RoboDK station: Trabajo_AndreaCasal.rdk

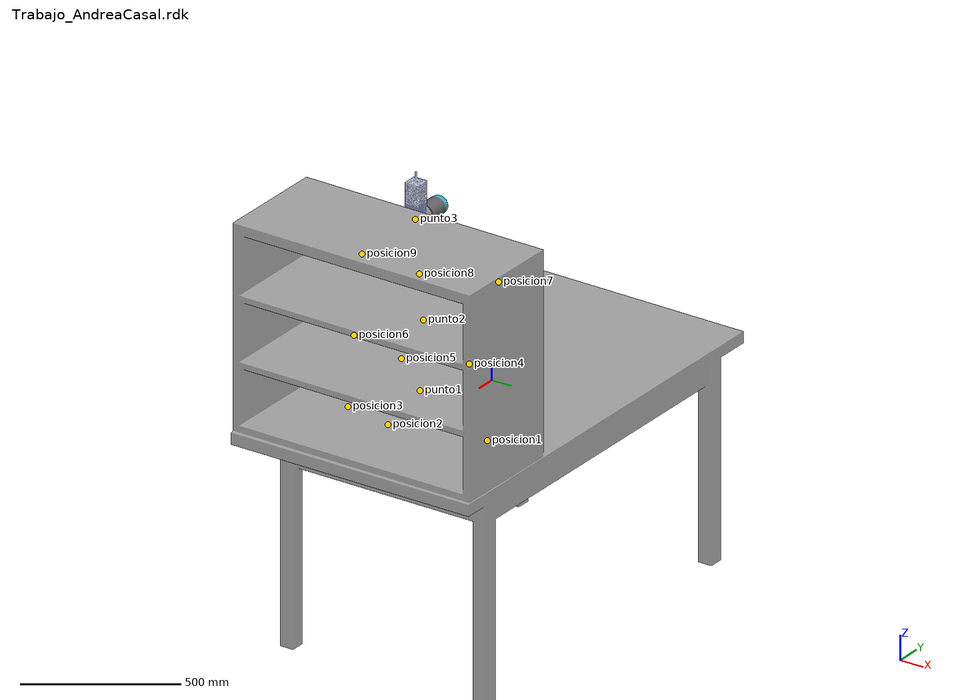
[picture v0: the station drawn from its stored meshes, robots at their saved joint values, targets as dots, program paths as lines]
Station Trabajo_AndreaCasal (saved by RoboDK 5.4.1). Poses are relative to the parent item; angles as X-Y-Z fixed-axis rotations.
  - frame UR3e Base at (447.56, 766.92, -5.55) mm, rotated rx 0 ry 0 rz -89.36 deg
    - robot UR3e: 6 axes, payload 3 kg, reach 500 mm, repeatability 0.03 mm, weight 11 kg
        modified DH rows (alpha deg, a mm, theta deg, d mm): 0, 0, 0, 151.9; 90, 0, 180, 0; 0, 243.55, 0, 0; 0, 213.2, 0, 131.05; -90, 0, 0, 85.35; 90, 0, 180, 92.1
        joint limits [-360, -360, -360, -360, -360, -360] to [360, 360, 360, 360, 360, 360]; home [0, -90, -90, 0, 90, 0]; saved at [-9.797, -78.984, -66.655, -34.361, 99.797, 0]
      - tool RGI-35-14-O-B, TCP at (0, 0, 3.37) mm, rotated rx 179.18 ry -0.35 rz -171.57 deg, size 50 x 211.5 x 50 mm, geometry from RGI-35-14-O-B.step
    - target punto1 (Cartesian target) at (291.92, -70.9, 62.1) mm, rotated rx 0 ry 0 rz -6.66 deg; joints [-219.826, -59.606, 132.901, -163.143, 270.876, 48.404] of UR3e
    - target punto2 (Cartesian target) at (275.14, -68.94, 300.54) mm, rotated rx 0 ry 0 rz -6.66 deg; joints [-221.915, -101.216, 99.747, -88.347, 270.87, 46.315] of UR3e
    - target punto3 (Cartesian target) at (200.73, -151.17, 596.64) mm, rotated rx -90.76 ry -8.43 rz 89.64 deg; joints [-9.797, -78.984, -66.655, -34.361, 99.797, 0] of UR3e
    - target posicion1 (Cartesian target) at (461.35, 299.35, 59.69) mm, rotated rx 0 ry 0 rz -96.24 deg; joints [46.918, -169.172, -22.416, -78.205, 89.136, 224.729] of UR3e
    - target posicion2 (Cartesian target) at (546.96, -17.63, 62.08) mm, rotated rx -0.01 ry 0.01 rz -96.16 deg; joints [12.113, 168.263, -333.534, 255.925, 89.422, 189.837] of UR3e
    - target posicion3 (Cartesian target) at (477.2, -215.05, 41.8) mm, rotated rx -1.06 ry 0.61 rz -88.34 deg; joints [-9.799, 157.17, -315.046, 247.588, 90.208, 160.103] of UR3e
    - target posicion4 (Cartesian target) at (440.56, 215.93, 293.67) mm, rotated rx 0 ry 0 rz -86.75 deg; joints [190.711, -24.384, -15.088, -51.292, -90.455, 179.024] of UR3e
    - target posicion5 (Cartesian target) at (502.45, 3.39, 277.35) mm, rotated rx 0 ry 0 rz -92.54 deg; joints [165.302, -24.016, -10.395, -56.461, -90.172, 159.416] of UR3e
    - target posicion6 (Cartesian target) at (449.26, -212.68, 277.35) mm, rotated rx 0 ry 0 rz -135.25 deg; joints [139.463, -20.178, -19.363, -51.244, -90.418, 176.285] of UR3e
    - target posicion7 (Cartesian target) at (348.61, 264.74, 553.8) mm, rotated rx -49.09 ry 85.03 rz -169.88 deg; joints [-170.394, -38.323, -15.462, -120.665, -41.22, -98.9] of UR3e
    - target posicion8 (Cartesian target) at (433.63, 23.76, 549.67) mm, rotated rx -48.02 ry 79.49 rz 134.2 deg; joints [-199.224, -34.418, -27.438, -110.141, -69.026, 266.448] of UR3e
    - target posicion9 (Cartesian target) at (396.78, -218.94, 536.56) mm, rotated rx 96.2 ry 89.06 rz -87.12 deg; joints [-14.289, -136.878, -4.448, -38.914, -259.855, 260.589] of UR3e
  - folder Entorno
    - object Pieza lego at (447.74, 637.94, 12.64) mm, rotated rx 1.86 ry 0 rz 0 deg, size 31.7 x 31.7 x 23.7 mm, geometry from LEGO_DUPLO_BRICK_2X2.igs
    - object Pieza lego 2 at (503.04, 474.4, 3.15) mm, size 31.7 x 31.7 x 23.7 mm, geometry from LEGO_DUPLO_BRICK_2X2.igs
    - object Mesa at (903.95, 87.57, -37.84) mm, rotated rx 90 ry 0 rz 90.24 deg, size 1500 x 750 x 900 mm, geometry from mesa(150x90).stl
    - object Estanteria at (0, 0, 0) mm, size 900 x 400 x 720 mm, geometry from estanteria.stl
  - Python program Programa (listed below)

--- Python program Programa ---
# LIBRERÍAS
from robodk import robolink    # RoboDK API
from robodk import robomath    # Robot toolbox
from tkinter import *
import threading
import random

# Para ser compatible con versiones antiguas de RoboDK:
from robodk import *      # RoboDK API
from robolink import *    # Robot toolbox

# ************************* FUNCIONES **********************************
# Función para cerrar la ventana
def onClose():
    ventana.destroy()
    RDK.Item('objeto').Delete()
    quit(0)

# Función para clasificar
def clasifica(clasificacion):
    # Posición inicial
    robot.MoveL(punto3)

    # Tarjet del objeto

    posObjeto = random.randint(1,3)
    if posObjeto == 1:
        objeto.setPose(transl(-500 ,0,50))
    if posObjeto == 2:
        objeto.setPose(transl(-500 ,200,50))
    if posObjeto == 3:
        objeto.setPose(transl(-500 ,-200,50))

    # Coger el objeto
    robot.MoveJ(objeto)
    robot.MoveJ(punto3)

    # Posición a la que debe mover el objeto en función de la clasificación:
    #Primera balda:
    if clasificacion == 1 or clasificacion == 2 or clasificacion == 3:

        robot.MoveL(punto1)

        if clasificacion == 1:
            robot.MoveL(posicion1)

        if clasificacion == 2:
            robot.MoveL(posicion2)

        if clasificacion == 3:
            robot.MoveL(posicion3)

        robot.MoveL(punto1)

    # Segunda balda:
    if clasificacion == 4 or clasificacion == 5 or clasificacion == 6:

        robot.MoveL(punto2)

        if clasificacion == 4:
            robot.MoveL(posicion4)

        if clasificacion == 5:
            robot.MoveL(posicion5)

        if clasificacion == 6:
            robot.MoveL(posicion6)

        robot.MoveL(punto2)

    # Tercera balda:
    if clasificacion == 7 or clasificacion == 8 or clasificacion == 9:

        robot.MoveL(punto3)

        if clasificacion == 7:
            robot.MoveL(posicion7)

        if clasificacion == 8:
            robot.MoveL(posicion8)

        if clasificacion == 9:
            robot.MoveL(posicion9)

        robot.MoveL(punto3)


# ************************ PROGRAMA ROBOT *****************************
# Link a RoboDK
RDK = robolink.Robolink()

# Escoger el objeto del robot, de la herramienta y la pieza lego:
robot = RDK.Item('', ITEM_TYPE_ROBOT)
frame = RDK.Item('UR3e Base',ITEM_TYPE_FRAME)
robot.setPoseFrame(frame)
obj = RDK.Item('Pieza lego')
tool = RDK.Item('RGI-35-14-O-B')
objeto = RDK.AddTarget('objeto', frame)


# Se cogen los tarjet
# Tarjet para los puntos de partida para los movimientos
punto1 = RDK.Item('punto1', ITEM_TYPE_TARGET)
punto2 = RDK.Item('punto2', ITEM_TYPE_TARGET)
punto3 = RDK.Item('punto3', ITEM_TYPE_TARGET)

# Tarjet para la colocación en las posiciones 1, 2 y 3 (primera balda)
posicion1 = RDK.Item('posicion1', ITEM_TYPE_TARGET)
posicion2 = RDK.Item('posicion2', ITEM_TYPE_TARGET)
posicion3 = RDK.Item('posicion3', ITEM_TYPE_TARGET)

# Tarjet para la colocación en las posiciones 4, 5 y 6 (segunda balda)
posicion4 = RDK.Item('posicion4', ITEM_TYPE_TARGET)
posicion5 = RDK.Item('posicion5', ITEM_TYPE_TARGET)
posicion6 = RDK.Item('posicion6', ITEM_TYPE_TARGET)

# Tarjet para la colocación en las posiciones 7, 8 y 9 (tercera balda)
posicion7 = RDK.Item('posicion7', ITEM_TYPE_TARGET)
posicion8 = RDK.Item('posicion8', ITEM_TYPE_TARGET)
posicion9 = RDK.Item('posicion9', ITEM_TYPE_TARGET)



# Create a new window
ventana = tkinter.Tk()
ventana.geometry("400x300")

# Fijar titulo de la ventana
ventanaTitulo = 'Clasificador'
ventana.title(ventanaTitulo)

# Se elimina la ventana al cerrarla
ventana.protocol("WM_DELETE_WINDOW", onClose)


# Se incrusta la ventana
#EmbedWindow(ventanaTitulo)
clasificacion = tkinter.IntVar()
opciones = [("1",1),
            ("2",2),
            ("3",3),
            ("4",4),
            ("5",5),
            ("6",6),
            ("7",7),
            ("8",8),
            ("9",9)]

for texto,valor in opciones:
    tkinter.Radiobutton(ventana,text=texto, variable=clasificacion, value=valor).pack()

# Se añade un boton (clasifica al pulsarlo)
botonClasifica = Button(ventana, text='Clasificar', height=5, width=8, command= lambda: clasifica(clasificacion.get()))
botonClasifica.pack(fill=X)

# Se lanza la ventana en bucle
ventana.mainloop()


# Terminar al acabar el movimiento
robot.RunInstruction('Program_Done')
